FUNCTION_BLOCK Komplett
VAR_INPUT
END_VAR
VAR_OUTPUT
END_VAR
VAR
	Timer1: TON;
END_VAR

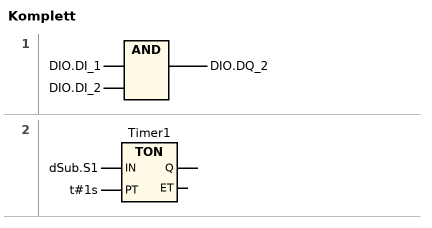
// NETWORK 1
DIO.DQ_2 := DIO.DI_1 AND DIO.DI_2;

// NETWORK 2
Timer1(IN := dSub.S1, PT := t#1s); // TON

END_FUNCTION_BLOCK

(* stored: Version 1.1.0.1, ProductVersion 3.1.4022.7
   POU Komplett: Id {1acb2216-9485-4b7b-a260-407b6101ea82}, SpecialFunc None *)
